Staubli VAL3: start.pgx

program start()
  local num l_nX
  local num l_nY
begin

  for l_nX = 0 to 2
    for l_nY = 0 to 3
      nMatrix1[l_nX,l_nY] = l_nX*l_nY
      nMatrix2[l_nX,l_nY] = l_nX+l_nY
    endFor
  endFor

  ? "Matrix 1:"
  call util:printNum2d(nMatrix1)
  ? "Matrix 2:"
  call util:printNum2d(nMatrix2)

  ? "test add: add(nMatrix1,nMatrix2, nResult)"
  call add(nMatrix1,nMatrix2, nResult)
  call util:printNum2d(nResult)


end
